PROGRAM MAIN
VAR
	Single:BOOL;
	Reset:bool;
	foto: BOOL;
	HaveResult:BOOL;
	Resultado: ARRAY [0..7] OF REAL;
END_VAR


GVL.FQM.SingleShot(Enable:=Single,Execute:=foto,Measurement => HaveResult, Results => Resultado);
GVL.FQM();

END_PROGRAM

(* stored: Version 1.1.0.1, ProductVersion 3.1.4024.9
   POU MAIN: Id {b79f9dd0-5a5a-4986-a3c7-739531a1facc}, SpecialFunc None *)
